VAR_GLOBAL
	
	qCylinderUp            				AT %Q*	 		: 	BOOL;
	qCylinderDown						AT %Q*	 		: 	BOOL;
	
	iCylinderUp            				AT %I*	 		: 	BOOL;
	iCylinderDown						AT %I*	 		: 	BOOL;

END_VAR

(* stored: Version 1.1.0.1, ProductVersion 3.1.4026.17
   GVL GVL_CylinderTest: Id {4e6ce3fe-25e3-4459-bcc0-aa2e161d9f33} *)
